Universal Robots PolyScope program: XMLRPC_loop.urp

Program XMLR PC_loop (installation=default directory=/home/ur/ursim-current/programs createdIn=3.1.16828 lastSavedIn=5.13.0 robotSerialNumber=20195399999)
Calibrated DH parameters: a=[0, -0.24355, -0.2132, 0, 0, 0]; d=[0.15185, 0, 0, 0.13105, 0.08535, 0.0921]; alpha=[1.570796, 0, 0, 1.570796, -1.570796, 0]; deltaTheta=[0, 0, 0, 0, 0, 0]
InitVariablesNode
BeforeStart
  camera := rpc_factory("xmlrpc","http://192.168.56.1:50000")
Robot Program (runOnlyOnce=false)
  Loop Forever
    next_pose := camera.get_next_pose(Joint_6_name)
    MoveJ speed 60 deg/s, acceleration 80 deg/s^2 (useActiveTCP=true) feature=Base
      Waypoint Variable (Variable): variable=next_pose
  Halt
  next_pose := camera.get_next_pose(Joint_6_name)
  MoveJ speed 60 deg/s, acceleration 80 deg/s^2 (useActiveTCP=true) feature=Base
    Waypoint Variable (Variable): variable=next_pose
